PROGRAM MAIN_CFC
VAR
	ProductionAnalytics		:	ProductionAnalytics;
	RawDataArray	: ARRAY[1..10] OF REAL := [5, 3, 8.3, 5, 6, 5, 5, 23, 5, 9];
	SortedArray		: ARRAY[1..10] OF REAL;
	
	Sort			: BOOL;
	GetMean			: BOOL;
	GetStdDev		: BOOL;
	GetTotal		: BOOL;
	GetMax			: BOOL;
	FindItem		: BOOL;
	Mean			: REAL;
	StdDev			: REAL;
	Total			: REAL;
	MaxItem			: REAL;
	FoundItemIdx	: UINT;
	ItemFound		: BOOL;
	ValidInput		: BOOL;
	IsSorted		: BOOL;
	ValueToFind		: REAL;
END_VAR

VAR CONSTANT
	ARRAY_SIZE		: UINT := 10;
END_VAR
VAR // added by the converter: edge detectors and wires of the graphical bodies
    _w1, _w2, _w3, _w4, _w5, _w6, _w7, _w8, _w9, _w10 : ANY;
END_VAR

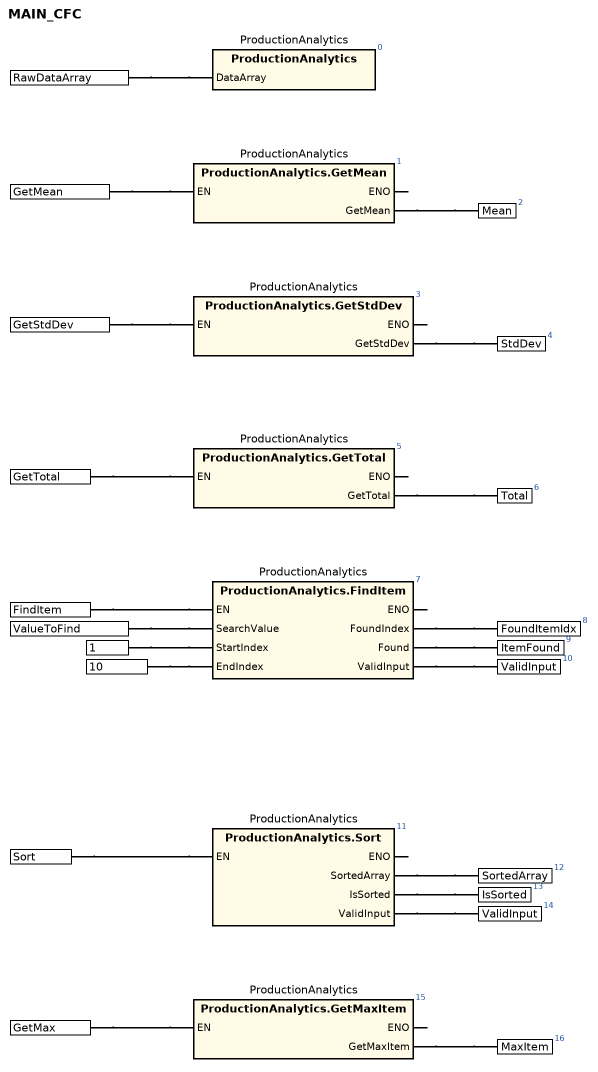
ProductionAnalytics(DataArray := RawDataArray);
IF GetMean THEN _w1 := ProductionAnalytics.GetMean(); END_IF
Mean := _w1;
IF GetStdDev THEN _w2 := ProductionAnalytics.GetStdDev(); END_IF
StdDev := _w2;
IF GetTotal THEN _w3 := ProductionAnalytics.GetTotal(); END_IF
Total := _w3;
IF FindItem THEN ProductionAnalytics.FindItem(SearchValue := ValueToFind, StartIndex := 1, EndIndex := 10, FoundIndex => _w4, Found => _w5, ValidInput => _w6); END_IF
FoundItemIdx := _w4;
ItemFound := _w5;
ValidInput := _w6;
IF Sort THEN ProductionAnalytics.Sort(SortedArray => _w7, IsSorted => _w8, ValidInput => _w9); END_IF
SortedArray := _w7;
IsSorted := _w8;
ValidInput := _w9;
IF GetMax THEN _w10 := ProductionAnalytics.GetMaxItem(); END_IF
MaxItem := _w10;

END_PROGRAM

(* stored: Version 1.1.0.1, ProductVersion 3.1.4024.15
   POU MAIN_CFC: Id {646714f0-3ce8-47b0-9b2a-f6dab68a5afc}, SpecialFunc None *)
